// LS Electric XG5000 project: PLC Coli Controll with Python
// PLC LSPLC

PROGRAM NewProgram (task: 스캔 프로그램)

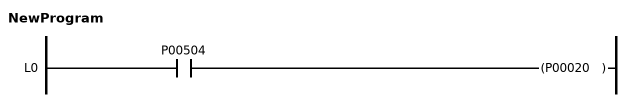
; L0
LOAD      P00504
OUT       P00020